// Mitsubishi GX Works2 project: neww (3)   PLC: FX3G
// New wworks

// global labels: Global1
VAR_GLOBAL CONSTANT
  FlourMin : REAL := 100.0;
END_VAR
VAR_GLOBAL
  FlourStock AT D1100 : REAL;
  aid1 AT M1 : BOOL;
  aid2 AT M2 : BOOL;
  YeastStock AT D1102 : REAL;
END_VAR
VAR_GLOBAL CONSTANT
  YeastMin : REAL := 20.0;
END_VAR
VAR_GLOBAL
  WaterStock AT D1104 : REAL;
END_VAR
VAR_GLOBAL CONSTANT
  WaterMin : REAL := 50.0;
END_VAR
VAR_GLOBAL
  OilStock AT D1106 : REAL;
END_VAR
VAR_GLOBAL CONSTANT
  OilMin : REAL := 30.0;
END_VAR
VAR_GLOBAL
  aid3 AT M3 : BOOL;
  aid4 AT M4 : BOOL;
  SpicesStock AT D1108 : REAL;
END_VAR
VAR_GLOBAL CONSTANT
  SpicesMin : REAL := 10.0;
END_VAR
VAR_GLOBAL
  aid5 AT M5 : BOOL;
  aid6 AT M6 : BOOL;
  StartBottom AT X010 : BOOL;
  aid7 AT M7 : BOOL;
  aod8 AT M8 : BOOL;
  workdaybolb AT Y010 : BOOL;
  Flour_Low AT M20 : BOOL;
  Yeast_Low AT M21 : BOOL;
  Water_Low AT M22 : BOOL;
  Oil_Low AT M23 : BOOL;
  Spices_Low AT M24 : BOOL;
  ResetBottom AT X007 : BOOL;
  aid9 AT M9 : BOOL;
  aid10 AT M10 : BOOL;
  aid8 AT M8 : BOOL;
END_VAR
VAR_GLOBAL CONSTANT
  delay0 : INT := 30;
END_VAR
VAR_GLOBAL
  Ts0 AT TS0 : BOOL;
  Ts1 AT TS1 : BOOL;
END_VAR
VAR_GLOBAL CONSTANT
  delay1 : INT := 5;
END_VAR
VAR_GLOBAL
  aid11 AT M11 : BOOL;
  aid12 AT M12 : BOOL;
  aid13 AT M13 : BOOL;
  Ts2 AT TS2 : BOOL;
  bolb1 AT Y005 : BOOL;
  Rawmaterials AT X002 : BOOL;
END_VAR
VAR_GLOBAL CONSTANT
  delay2 : INT := 30;
END_VAR
VAR_GLOBAL
  kneading AT X001 : BOOL;
  Endkneading AT Y001 : BOOL;
  Swelling AT X011 : BOOL;
  Counter1 AT CC0 : BOOL;
END_VAR
VAR_GLOBAL CONSTANT
  count1 : WORD := 2;
END_VAR
VAR_GLOBAL
  Ts3 AT TS3 : BOOL;
END_VAR
VAR_GLOBAL CONSTANT
  delay3 : INT := 30;
END_VAR
VAR_GLOBAL
  aid14 AT M14 : BOOL;
  Ts4 AT TS4 : BOOL;
END_VAR
VAR_GLOBAL CONSTANT
  delay4 : INT := 5;
END_VAR
VAR_GLOBAL
  bolb2 AT Y003 : BOOL;
  Ts5 AT TS5 : BOOL;
END_VAR
VAR_GLOBAL CONSTANT
  delay5 : INT := 5;
END_VAR
VAR_GLOBAL
  bolb3 AT Y002 : BOOL;
  aid15 AT M15 : BOOL;
  aid16 AT M16 : BOOL;
  Ts6 AT TS6 : BOOL;
END_VAR
VAR_GLOBAL CONSTANT
  delay6 : INT := 40;
END_VAR
VAR_GLOBAL
  bolb4 AT Y004 : BOOL;
  Analogcheck AT X003 : BOOL;
  AnalogImput1 AT D1110 : REAL;
  AnalogImput2 AT D1112 : REAL;
END_VAR
VAR_GLOBAL CONSTANT
  minAnalog : REAL := 1.0;
  maxAnalog : REAL := 5.0;
END_VAR
VAR_GLOBAL
  aid17 AT M17 : BOOL;
  Counter2 AT CC1 : BOOL;
END_VAR
VAR_GLOBAL CONSTANT
  count2 : WORD := 2;
END_VAR
VAR_GLOBAL
  aid18 AT M18 : BOOL;
  aid19 AT M19 : BOOL;
  Ts7 AT TS7 : BOOL;
END_VAR
VAR_GLOBAL CONSTANT
  delay7 : INT := 50;
END_VAR
VAR_GLOBAL
  bolb5 AT Y006 : BOOL;
END_VAR

// task Task_01 (event TRUE, interval 0, priority 31): POU_01

PROGRAM POU_01
(* structured ladder/FBD written out as ST: instructions are called as NAME(EN, inputs, outputs); _pN, _eN, _tN stand for wires *)
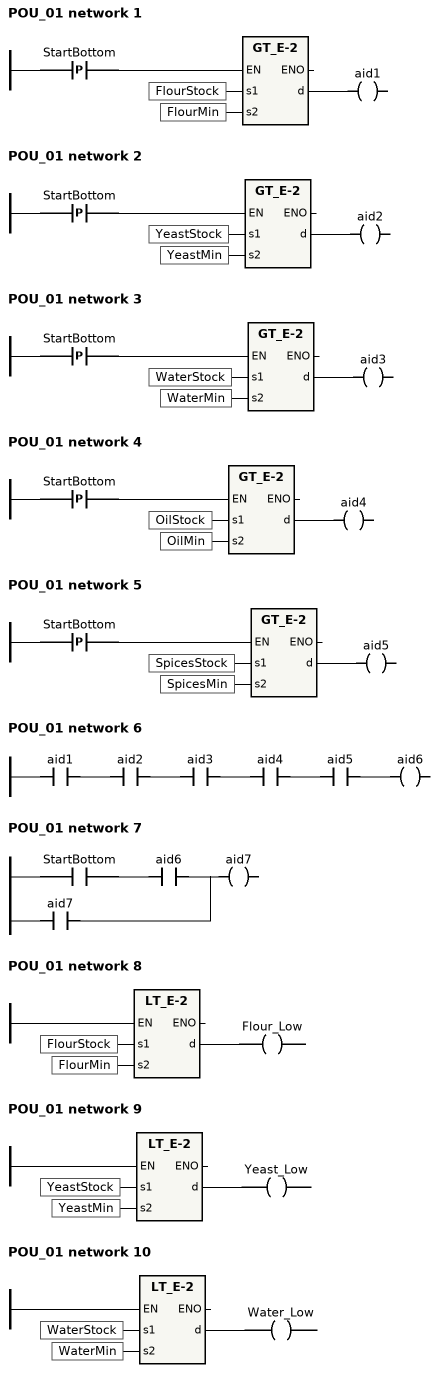
(* network 1 *)
GT_E(LDP(TRUE, StartBottom), FlourStock, FlourMin, _t1);
aid1 := _t1;
(* network 2 *)
GT_E(LDP(TRUE, StartBottom), YeastStock, YeastMin, _t1);
aid2 := _t1;
(* network 3 *)
GT_E(LDP(TRUE, StartBottom), WaterStock, WaterMin, _t1);
aid3 := _t1;
(* network 4 *)
GT_E(LDP(TRUE, StartBottom), OilStock, OilMin, _t1);
aid4 := _t1;
(* network 5 *)
GT_E(LDP(TRUE, StartBottom), SpicesStock, SpicesMin, _t1);
aid5 := _t1;
(* network 6 *)
aid6 := aid1 AND aid2 AND aid3 AND aid4 AND aid5;
(* network 7 *)
aid7 := (StartBottom AND aid6) OR aid7;
(* network 8 *)
LT_E(TRUE, FlourStock, FlourMin, _t1);
Flour_Low := _t1;
(* network 9 *)
LT_E(TRUE, YeastStock, YeastMin, _t1);
Yeast_Low := _t1;
(* network 10 *)
LT_E(TRUE, WaterStock, WaterMin, _t1);
Water_Low := _t1;
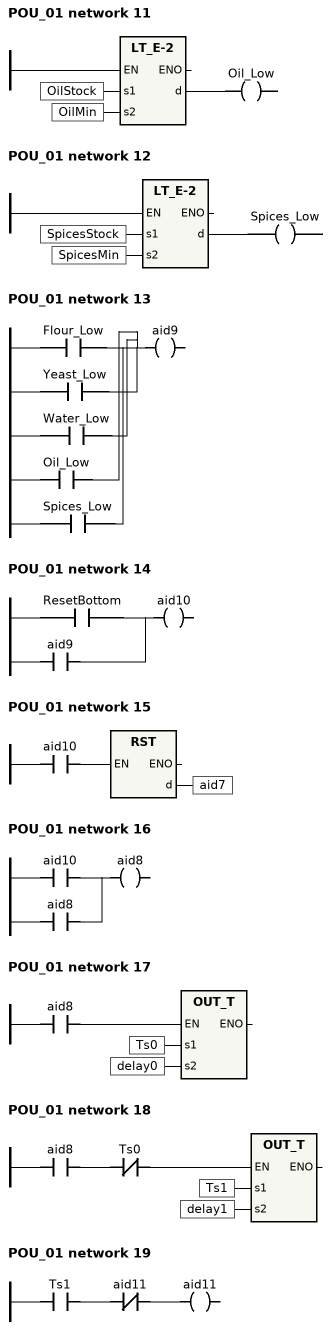
(* network 11 *)
LT_E(TRUE, OilStock, OilMin, _t1);
Oil_Low := _t1;
(* network 12 *)
LT_E(TRUE, SpicesStock, SpicesMin, _t1);
Spices_Low := _t1;
(* network 13 *)
aid9 := Flour_Low OR Yeast_Low OR Water_Low OR Oil_Low OR Spices_Low;
(* network 14 *)
aid10 := ResetBottom OR aid9;
(* network 15 *)
RST(aid10, aid7);
(* network 16 *)
aid8 := aid10 OR aid8;
(* network 17 *)
OUT_T(aid8, Ts0, delay0);
(* network 18 *)
OUT_T(aid8 AND NOT Ts0, Ts1, delay1);
(* network 19 *)
aid11 := Ts1 AND NOT aid11;
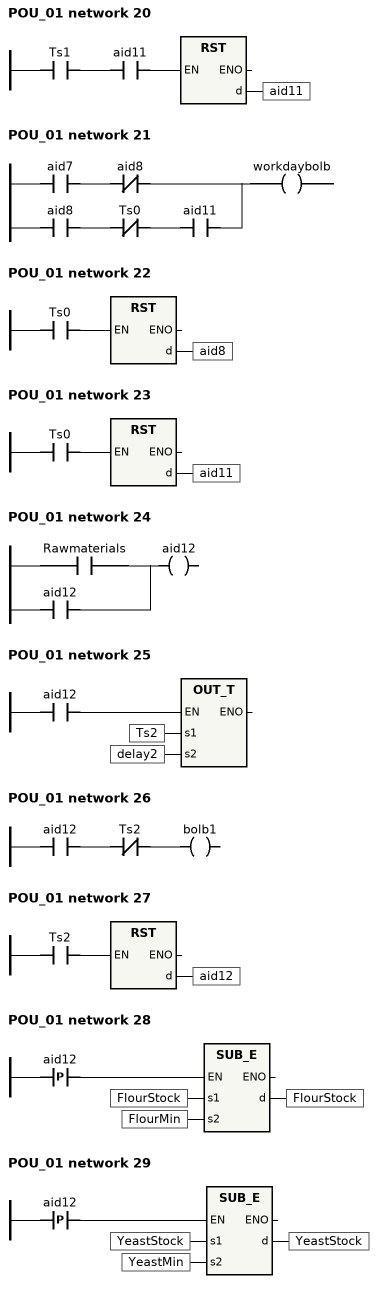
(* network 20 *)
RST(Ts1 AND aid11, aid11);
(* network 21 *)
workdaybolb := (aid7 AND NOT aid8) OR (aid8 AND NOT Ts0 AND aid11);
(* network 22 *)
RST(Ts0, aid8);
(* network 23 *)
RST(Ts0, aid11);
(* network 24 *)
aid12 := Rawmaterials OR aid12;
(* network 25 *)
OUT_T(aid12, Ts2, delay2);
(* network 26 *)
bolb1 := aid12 AND NOT Ts2;
(* network 27 *)
RST(Ts2, aid12);
(* network 28 *)
SUB_E(LDP(TRUE, aid12), FlourStock, FlourMin, FlourStock);
(* network 29 *)
SUB_E(LDP(TRUE, aid12), YeastStock, YeastMin, YeastStock);
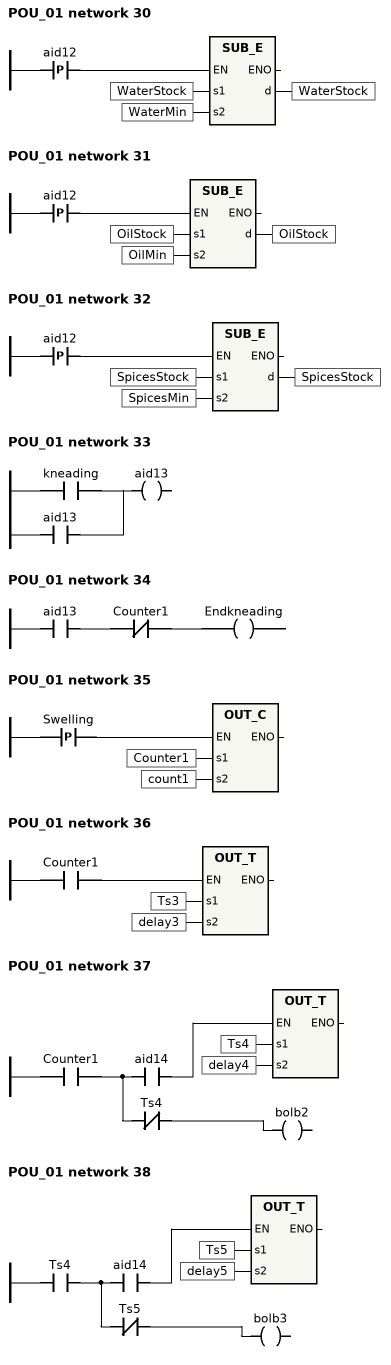
(* network 30 *)
SUB_E(LDP(TRUE, aid12), WaterStock, WaterMin, WaterStock);
(* network 31 *)
SUB_E(LDP(TRUE, aid12), OilStock, OilMin, OilStock);
(* network 32 *)
SUB_E(LDP(TRUE, aid12), SpicesStock, SpicesMin, SpicesStock);
(* network 33 *)
aid13 := kneading OR aid13;
(* network 34 *)
Endkneading := aid13 AND NOT Counter1;
(* network 35 *)
OUT_C(LDP(TRUE, Swelling), Counter1, count1);
(* network 36 *)
OUT_T(Counter1, Ts3, delay3);
(* network 37 *)
OUT_T(Counter1 AND aid14, Ts4, delay4);
bolb2 := Counter1 AND NOT Ts4;
(* network 38 *)
OUT_T(Ts4 AND aid14, Ts5, delay5);
bolb3 := Ts4 AND NOT Ts5;
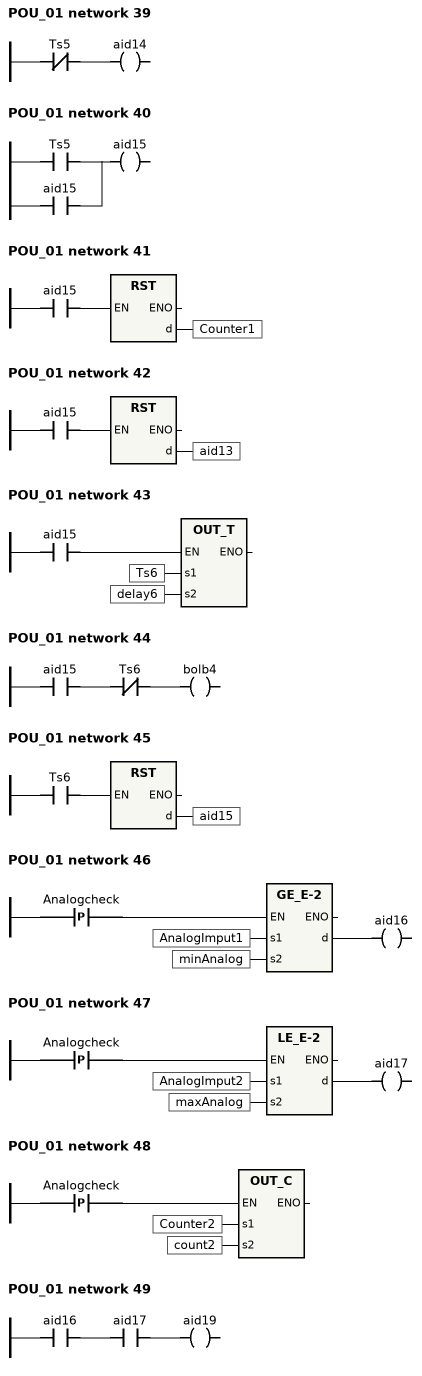
(* network 39 *)
aid14 := NOT Ts5;
(* network 40 *)
aid15 := Ts5 OR aid15;
(* network 41 *)
RST(aid15, Counter1);
(* network 42 *)
RST(aid15, aid13);
(* network 43 *)
OUT_T(aid15, Ts6, delay6);
(* network 44 *)
bolb4 := aid15 AND NOT Ts6;
(* network 45 *)
RST(Ts6, aid15);
(* network 46 *)
GE_E(LDP(TRUE, Analogcheck), AnalogImput1, minAnalog, _t1);
aid16 := _t1;
(* network 47 *)
LE_E(LDP(TRUE, Analogcheck), AnalogImput2, maxAnalog, _t1);
aid17 := _t1;
(* network 48 *)
OUT_C(LDP(TRUE, Analogcheck), Counter2, count2);
(* network 49 *)
aid19 := aid16 AND aid17;
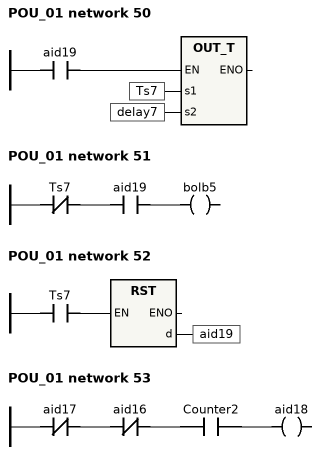
(* network 50 *)
OUT_T(aid19, Ts7, delay7);
(* network 51 *)
bolb5 := NOT Ts7 AND aid19;
(* network 52 *)
RST(Ts7, aid19);
(* network 53 *)
aid18 := NOT aid17 AND NOT aid16 AND Counter2;
END_PROGRAM
